(* PLC project CoDeSys External Library Template, WAGO e!COCKPIT e!COCKPIT, author 3S - Smart Software Solutions GmbH *)
(* stored: creationDateTime 2019-10-29T14:38:30.5385009, version 3.5.5.30, modificationDateTime 2019-10-29T14:38:06.5373783, organization 3S - Smart Software Solutions GmbH *)
(* Library project template with all possible element types, docu and a sample project structure *)

(* Autor: Paweł Kąkol, 2018-09-04-PK Prawa majątkowe: Solwena Sp. z o.o., Aktualizacje: 2019-02-18-AWy: alarm braku zmiany wartości napięcia lub prądu, zmiana klas alarmów Opis: fb służy do definicji klasy alarmów w fb analizatora sieci ECA0 na budynkach PPP Sopot (ENGIE) Diris A40 *)
{attribute 'qualified_only'}
{attribute 'strict'}
TYPE enumPPPSAnalizatorDirisA40ErrorKlasa : (BrakKomunikacji := enumKlasaAlarmu.AwariaAutomatyki, BrakZmianyParametrow := enumKlasaAlarmu.AwariaAutomatyki);
END_TYPE
